FUNCTION_BLOCK FB_ValveMaskHandler
VAR_INPUT
    abValveMaskSetRequest : BOOL; // single ATEQ: request/ack from ATEQ handler
    aValveMaskSteps       : ARRAY[0..GVL_AteqConfig.nMaxTestSteps - 1] OF ST_ValveMaskStep;
    aAteqValveMask        : ARRAY[0..3] OF DWORD; // next/target mask (4 DWORDs)
END_VAR

VAR_OUTPUT
    bValveMaskSetDone     : BOOL;
    aCurrentValveMask     : ARRAY[0..3] OF DWORD; // currently applied mask (to FB_ValveIo)
    nCurrentSeqStepIndex  : INT;
END_VAR

VAR
    eState                : (IDLE, TRANSITION_HOLD, APPLY_FINAL);

    aPreviousMask         : ARRAY[0..3] OF DWORD;
    aIntermediateMask     : ARRAY[0..3] OF DWORD; // phase-A mask (applied during hold)

    tTransitionHold       : TON;
    bTransitionTimerStarted : BOOL;

    i                     : INT;
    stSeqCurrentStep                  : ST_ValveMaskStep; // local alias
END_VAR

// This FB is called by each FB_ValveIo instances.
// Every ATEQ device will have the dedicated set of ValveBanks or IOBlocks, therefor FB_ValveMaskHandler must be instantiated per ATEQ device.
// Mask sorting always starts at Slot0 , no offsetting or indexing needed.

stSeqCurrentStep := aValveMaskSteps[nCurrentSeqStepIndex]; // Step check may be removed to higher level recipe handler (FB_SequenceStepsHandler)

// Step readiness check (single ATEQ)
    IF NOT abValveMaskSetRequest THEN
			bValveMaskSetDone := FALSE;	// not ready
        RETURN; // skip state machine until the request is present
    END_IF


CASE eState OF

    IDLE:
        aPreviousMask := aCurrentValveMask;

        CASE stSeqCurrentStep.eTransitionMode OF

            Immediate:
                aCurrentValveMask := aAteqValveMask;
                bValveMaskSetDone := TRUE;
                nCurrentSeqStepIndex := nCurrentSeqStepIndex + 1;

            HoldPrevious_ON: // OBC (Open Before Close)
                // Phase A: open next while keeping previous
                FOR i := 0 TO 3 DO
                    aIntermediateMask[i] := aPreviousMask[i] OR aAteqValveMask[i];
                    aCurrentValveMask[i] := aIntermediateMask[i];
                END_FOR

                bTransitionTimerStarted := FALSE;
                tTransitionHold(IN := FALSE); // ensure timer is reset
                bValveMaskSetDone := FALSE;
                eState := TRANSITION_HOLD;

            HoldNext_OFF: // CBO (Close Before Open)
                // Phase A: close any conflicting bits first (keep previous but clear any bits that are in next)
                FOR i := 0 TO 3 DO
                    aIntermediateMask[i] := aPreviousMask[i] AND NOT aAteqValveMask[i];
                    aCurrentValveMask[i] := aIntermediateMask[i];
                END_FOR
                // prepare timer
                bTransitionTimerStarted := FALSE;
                tTransitionHold(IN := FALSE);
                bValveMaskSetDone := FALSE;
                eState := TRANSITION_HOLD;

        END_CASE

    TRANSITION_HOLD:
        // Start the timer on the first cycle in this state with edge
        IF NOT bTransitionTimerStarted THEN
            tTransitionHold(IN := TRUE, PT := aValveMaskSteps[nCurrentSeqStepIndex].tTransitionHoldTime);
            bTransitionTimerStarted := TRUE;
        ELSE
            tTransitionHold(IN := TRUE); // Keep timer running
        END_IF

        // While in hold, aCurrentValveMask remains the intermediateMask (already set)
        IF tTransitionHold.Q THEN
            // apply final mask
            // Stop timer and clear flag
            tTransitionHold(IN := FALSE);
            bTransitionTimerStarted := FALSE;
            eState := APPLY_FINAL;
        END_IF

    APPLY_FINAL:
        // Final application: set the target mask
        FOR i := 0 TO 3 DO
            aCurrentValveMask[i] := aAteqValveMask[i];
        END_FOR
        bValveMaskSetDone := TRUE;
        // Advance sequence index
        nCurrentSeqStepIndex := nCurrentSeqStepIndex + 1;
        // return to IDLE
        eState := IDLE;

END_CASE

METHOD M_old : BOOL
VAR_INPUT
    abValveMaskSetRequest : BOOL; // Single ATEQ handler, just one flag
    aValveMaskSteps       : ARRAY[0..GVL_AteqConfig.nMaxTestSteps - 1] OF ST_ValveMaskStep;
    aAteqValveMask        : ARRAY[0..3] OF DWORD; // Up to 128 valves for each ATEQ
END_VAR

VAR_OUTPUT
    bValveMaskSetDone     : BOOL;
    aCurrentValveMask     : ARRAY[0..3] OF DWORD; // Output mask (to valve IO block)
    nCurrentSeqStepIndex  : INT;
END_VAR

VAR
    bStepReady            : BOOL;
    tTransitionHold       : TON;
    eState                : IDLE, TRANSITION_HOLD, APPLY_FINAL;
    aPreviousMask         : ARRAY[0..3] OF DWORD;
    aIntermediateMask     : ARRAY[0..3] OF DWORD;
    i                     : UINT;
END_VAR
// This FB is called by each FB_ValveIo instances.
// Every ATEQ device will have the dedicated set of ValveBanks or IOBlocks, therefor FB_ValveMaskHandler must be instantiated per ATEQ device.
// Mask sorting always starts at Slot0 , no offsetting or indexing needed.


bStepReady := TRUE;	// Step readiness check

IF (aValveMaskSteps[nCurrentSeqStepIndex].nExpectedDoneMask <> 0) THEN
    IF NOT abValveMaskSetRequest THEN
        bStepReady := FALSE;
    END_IF
END_IF


CASE eState OF

    IDLE:
        IF bStepReady THEN
            aPreviousMask := aCurrentValveMask;

            CASE aValveMaskSteps[nCurrentSeqStepIndex].eTransitionMode OF

                HoldPrevious_ON: // OBC Open Next before Closing Previous
                    aIntermediateMask := aAteqValveMask;
                    FOR i := 0 TO 3 DO
                        aCurrentValveMask[i] := aPreviousMask[i] OR aIntermediateMask[i];
                    END_FOR
                    eState := TRANSITION_HOLD;

                HoldNext_OFF: // CBO Close Previous before Opening Next
                    aIntermediateMask := aAteqValveMask;
                    FOR i := 0 TO 3 DO
                        aCurrentValveMask[i] := aPreviousMask[i] AND NOT aIntermediateMask[i];
                    END_FOR
                    eState := TRANSITION_HOLD;

                Immediate:
                    aCurrentValveMask := aAteqValveMask;
                    bValveMaskSetDone := TRUE;
                    nCurrentSeqStepIndex := nCurrentSeqStepIndex + 1;
            END_CASE
        END_IF

    TRANSITION_HOLD:
        tTransitionHold(IN := TRUE, PT := aValveMaskSteps[nCurrentSeqStepIndex].tTransitionHoldTime);
        IF tTransitionHold.Q THEN
            eState := APPLY_FINAL;
            tTransitionHold(IN := FALSE);
        END_IF

    APPLY_FINAL:
        aCurrentValveMask := aAteqValveMask;
        bValveMaskSetDone := TRUE;
        nCurrentSeqStepIndex := nCurrentSeqStepIndex + 1;
        eState := IDLE;

END_CASE
END_METHOD

END_FUNCTION_BLOCK

(* stored: Version 1.1.0.1
   POU FB_ValveMaskHandler: Id {852b63b7-129e-4d4e-b0a2-86d27375b5d0}, SpecialFunc None
   Method M_old: Id {35ed2413-461b-4b06-894b-5bfbb898bd34} *)
